INTERFACE I_Module

END_INTERFACE

(* stored: Version 1.1.0.1, ProductVersion 3.1.4024.15
   Itf I_Module: Id {94b91e81-af3e-49aa-a70a-2d93c908d3be} *)
